Staubli VAL3: Control_PanelD.pgx

public program Control_PanelD()
begin

  //默认两个框
  call Control_PanelS("",20,0,18,11)


end
